TYPE ST_IO2_Diagnostic :
STRUCT
	bState		: BOOL;
	sVarName		: STRING;

END_STRUCT
END_TYPE

(* stored: Version 1.1.0.1
   DUT ST_IO2_Diagnostic: Id {c4da3994-b704-4b31-beba-c2b3c94190d1} *)
